PROGRAM P4_02_Read
VAR
	fbDBRead    	:FB_PLCDBCmdEvt(sNetID:=CONST.AMS_NETID, tTimeout:=DEFAULT_ADS_TIMEOUT);
	
	tableColumns	:ARRAY [0..5] OF STRING(50) := ['DateTime', 'User', 'Event', 'Description', 'OldValue', 'NewValue'];
	arrParam		:ARRAY [0..5] OF ST_ExpParameter := [(sParaName := 'DateTime', nParaSize := 4, eParaType := E_EXPPARAMETERTYPE.DateTime), 
														(sParaName := 'User', nParaSize := 101, eParaType := E_EXPPARAMETERTYPE.STRING_), 
														(sParaName := 'Event', nParaSize := 101, eParaType := E_EXPPARAMETERTYPE.STRING_), 
														(sParaName := 'Description', nParaSize := 101, eParaType := E_EXPPARAMETERTYPE.STRING_), 
														(sParaName := 'OldValue', nParaSize := 101, eParaType := E_EXPPARAMETERTYPE.STRING_), 
														(sParaName := 'NewValue', nParaSize := 101, eParaType := E_EXPPARAMETERTYPE.STRING_)];
	stRecord		:ARRAY[0..999] OF ST_AuditTrail;	
	
	stDBParam 		:ST_AuditTrail;	
	nRecords		:UDINT;
	sCmd			:STRING[300];

END_VAR
VAR // added by the converter: edge detectors and wires of the graphical bodies
    _w1 : BOOL;
END_VAR

//**************HMI FILTER - COMPOSE QUERY***************
sCmd:='SELECT * FROM `audit_trail`';
IF GV.stHMI.stAudit_Ctrl.bFilter THEN
	
	IF GV.stHMI.stAudit_Ctrl.enFilter_Event <> 0 THEN
		sCmd:=CONCAT(sCmd,'WHERE `Event` = $'');
		sCmd:=CONCAT(sCmD,TO_STRING(GV.stHMI.stAudit_Ctrl.enFilter_Event));
		sCmd:=CONCAT(sCmd,'$'');
	END_IF
	IF GV.stHMI.stAudit_Ctrl.sFilter_User <> GV.sEmptyString THEN
		IF GV.stHMI.stAudit_Ctrl.enFilter_Event = 0 THEN
			sCmd:=CONCAT(sCmd,'WHERE `User` LIKE $'%');
		ELSE
			sCmd:=CONCAT(sCmd,'AND `User` LIKE $'%');
		END_IF
		sCmd:=CONCAT(sCmD,GV.stHMI.stAudit_Ctrl.sFilter_User);
		sCmd:=CONCAT(sCmd,'$'');
	END_IF
	IF GV.stHMI.stAudit_Ctrl.sFilter_Key <> GV.sEmptyString THEN
		IF GV.stHMI.stAudit_Ctrl.enFilter_Event = 0 AND GV.stHMI.stAudit_Ctrl.sFilter_User = GV.sEmptyString THEN
			sCmd:=CONCAT(sCmd,'WHERE `Description` LIKE $'%');
		ELSE
			sCmd:=CONCAT(sCmd,'AND `Description` LIKE $'%');
		END_IF
		sCmd:=CONCAT(sCmD,GV.stHMI.stAudit_Ctrl.sFilter_Key);
		sCmd:=CONCAT(sCmd,'%$'');
	END_IF
	IF GV.stHMI.stAudit_Ctrl.dtFilter_From <> GV.stHMI.stAudit_Ctrl.dtFilter_To THEN
		IF GV.stHMI.stAudit_Ctrl.enFilter_Event = 0 AND GV.stHMI.stAudit_Ctrl.sFilter_User = GV.sEmptyString AND GV.stHMI.stAudit_Ctrl.sFilter_Key = GV.sEmptyString THEN
				sCmd:=CONCAT(sCmd,'WHERE `DateTime` BETWEEN $'');
			ELSE
				sCmd:=CONCAT(sCmd,'AND `DateTime` BETWEEN $'');
			END_IF
			sCmd:=CONCAT(sCmd,RIGHT(DT_TO_STRING(GV.stHMI.stAudit_Ctrl.dtFilter_From),19));
			sCmd:=CONCAT(sCmd,'$' AND $'');
			sCmd:=CONCAT(sCmd,RIGHT(DT_TO_STRING(GV.stHMI.stAudit_Ctrl.dtFilter_To),19));
			sCmd:=CONCAT(sCmd,'$'');
	END_IF
	GV.stTX_Python.sAuditExportQuery:=sCmd;
END_IF
sCmd:=CONCAT(sCmd,' ORDER BY `DateTime` DESC');


ACT_Cmd();

ACTION ACT_Cmd:
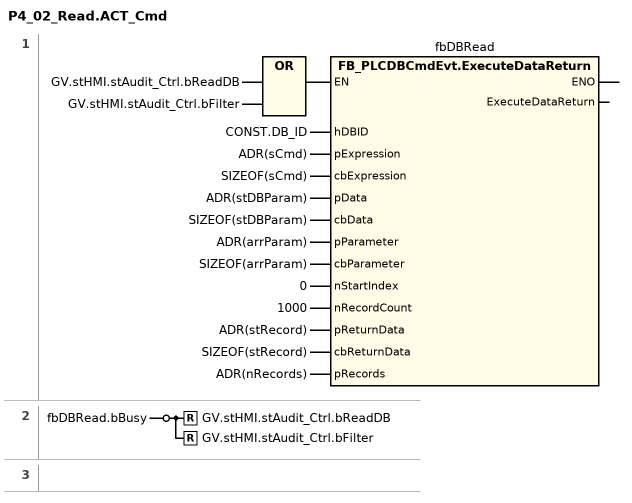
// NETWORK 1
IF GV.stHMI.stAudit_Ctrl.bReadDB OR GV.stHMI.stAudit_Ctrl.bFilter THEN
    fbDBRead.ExecuteDataReturn(
        hDBID := CONST.DB_ID,
        pExpression := ADR(sCmd),
        cbExpression := SIZEOF(sCmd),
        pData := ADR(stDBParam),
        cbData := SIZEOF(stDBParam),
        pParameter := ADR(arrParam),
        cbParameter := SIZEOF(arrParam),
        nStartIndex := 0,
        nRecordCount := 1000,
        pReturnData := ADR(stRecord),
        cbReturnData := SIZEOF(stRecord),
        pRecords := ADR(nRecords));
END_IF

// NETWORK 2
_w1 := NOT fbDBRead.bBusy;
GV.stHMI.stAudit_Ctrl.bReadDB R= _w1;
GV.stHMI.stAudit_Ctrl.bFilter R= _w1;

// NETWORK 3
END_ACTION

END_PROGRAM

(* stored: Version 1.1.0.1, ProductVersion 3.1.4024.13
   POU P4_02_Read: Id {b9f427ab-f48f-4ea1-a314-075d2a188de9}, SpecialFunc None
   Action ACT_Cmd: Id {3e7686b0-3678-4fe5-ab28-ae421e7557c5} *)
